(* IEC 61131-3 sources: std_i2980_v2.06_cp053/Source/IMM/ieccontrol/system (part 3) *)

(* ---- ABRuntimeMonitoring.pu ---- *)
(*
@h    ! WARNING !
@h    The Kemro K2 system (including software) only meets category B according to EN 954-1,
@h    thus it is not intended for usage in safety-relevant control applications in the field
@h    of personal safety (e.g. emergency stop).
@h    To implement potentially necessary safety-relevant control tasks, always use additional
@h    external safety devices that are intended for the particular purpose, and meet the necessary
@h    functional safety.
@h    For further information see EN 954-1 (EN ISO 13849-1) and/or the K2-x00 user manual, chapter
@h    "CE conformity, directives and standards".

This AB reacts on changes of sv_DataState and ODC1.sv_iInitOk
If sv_DataState is not nReady (this means reading or writing of data is in progress),
the runtime monitoring of the IEC - tasks will be switched off.
After sv_DataState changes to nReady again, the runtime monitoring will be switched on.
If the IEC - project is executed on Windows the runtime monitoring is switched off all the time.
The creation of the machine sequence, calculation of safety conditions, .... runs in TaskMid
To avoid cycle overflows during this procedure, the supervision is set to a higher value
during sequence creation.
Attention:
The supervision of TaskMid during creation of sequence should not be disabled so that
endless loops can be detected.
*)

IMPORT_OVER_LISTFILE
 SET_MAXIMUM_ACTIVE_INTERVAL
, tnDataState
, KCAT_HandleData
, KCAT_Status
, KSYS_Status

END_IMPORT

ALGORITHM_BLOCK ABRuntimeMonitoring #DUMMY_EDIT_BLOCK

SYSTEM_VAR
 sv_DataState : tnDataState (* indicates the state of xml handling (set by hmi) *);
 sv_bInitDone : BOOL;
 sv_bAllPUTasksExecuted : BOOL;
 sv_bInitStart : BOOL;
 sv_iActiveParamTransfers : DINT (* number of actually active parameter transfers (written by ABDriveParam.pu) *);
 sv_iReadMachineDataCount : UDINT (* counter which is increased after every loading of machine data  *);
 sv_iReadMoldDataCount : UDINT (* counter which is increased after every loading of mold data  *);
END_VAR

SYSTEM_OBJECT
 TaskException : TASK;
 TaskInject : TASK;
 TaskAnalog : TASK;
 TaskMid : TASK;
 TaskSequencer : TASK;
 PU_Task_13 : TASK;
 PU_Task_7 : TASK;
 PU_Task_3 : TASK;
 EV_Task_3 : TASK;
 EV_Task_7 : TASK;
 TaskHeating : TASK;
END_OBJECT

VAR
 mpiSequenceCreateState : REFTO DINT (* 0 nothing initialized, 10 sequence array initialized, 20 sequence array + safety initialized *);
 mbTaskPU13 : BOOL := FALSE;
 mbTaskPU7 : BOOL := FALSE;
 mbTaskPU3 : BOOL := FALSE;
 mbTaskEV3 : BOOL := FALSE;
 mbTaskEV7 : BOOL := FALSE;
END_VAR

POSTUPDATE_ALGORITHM pActivateDeactivate ON TaskException WITH sv_DataState,sv_bInitDone,mpiSequenceCreateState^,sv_iActiveParamTransfers

VAR
 StatusName : KCAT_HandleData;
 Name : STRING(255);
 Status : KCAT_Status;
 sValue : STRING(255);
 bIsWinNT : BOOL;
 bInitDone : BOOL;
 state : KSYS_Status;
 dSetInterval : TIME;
 bODC : BOOL;
 dSetTrigger : DINT;
END_VAR
#BEGIN_EDIT_BLOCK
(**************************************** WARNING ********************************************
 *** The KEBA Kemro K2 System including software is not intended for safety control tasks! ***
 ***                       For further information see Comment tab!                        ***
 *********************************************************************************************)

IF NOT bInitDone THEN
   Name := 'UOS.System';
   StatusName := KCAT_GetHandle(Name);
   IF StatusName.Status = KCAT_Status_OK THEN
      Status := KCAT_GetValue(Handle := StatusName.Handle, Buffer := sValue);
      IF (sValue = 'WINNT') THEN
         bIsWinNT := TRUE;
      ELSE
         bIsWinNT := FALSE;
      END_IF;
   END_IF;

   //get reference to state variable of sequence creation
   mpiSequenceCreateState := GET_SYNC_REFTO('ODC1.sv_iInitOK', T#0s, state);
   bODC := (state = KSYS_Status_OK);

   bInitDone := TRUE;
END_IF;

IF bIsWinNT THEN
   //don´t activate runtime monitoring if application is running on a pc
   RETURN;
END_IF;

IF bODC AND (mpiSequenceCreateState^ <> 20) THEN
   //creating of sequence in progress
   //creation of sequence, calculation of safety conditions, .... runs in TaskMid
   //-> set supervision to a higher value to avoid cycle overflows
   //supervision of TaskMid should not be disabled to detect endless loops
   dSetInterval := SET_MAXIMUM_ACTIVE_INTERVAL(TaskInject, GET_TASK_INTERVAL(TaskInject) * 10);
   dSetInterval := SET_MAXIMUM_ACTIVE_INTERVAL(TaskAnalog, GET_TASK_INTERVAL(TaskAnalog) * 10);
   dSetInterval := SET_MAXIMUM_ACTIVE_INTERVAL(TaskSequencer, GET_TASK_INTERVAL(TaskSequencer) * 10);
   dSetInterval := SET_MAXIMUM_ACTIVE_INTERVAL(TaskMid, GET_TASK_INTERVAL(TaskMid) * 200);

ELSIF sv_DataState <> nReady THEN
   //deactivate task runtime monitoring
   //if reading or writing of data is in progress
   dSetInterval := SET_MAXIMUM_ACTIVE_INTERVAL(TaskInject, T#0ms);
   dSetInterval := SET_MAXIMUM_ACTIVE_INTERVAL(TaskAnalog, T#0ms);
   dSetInterval := SET_MAXIMUM_ACTIVE_INTERVAL(TaskSequencer, T#0ms);
   dSetInterval := SET_MAXIMUM_ACTIVE_INTERVAL(TaskMid, T#0ms);

ELSIF sv_iActiveParamTransfers > 0 THEN
   //at least one paramter transfer is in progress -> increase maximum active interval of TaskMid
   dSetInterval := SET_MAXIMUM_ACTIVE_INTERVAL(TaskInject, GET_TASK_INTERVAL(TaskInject) * 10);
   dSetInterval := SET_MAXIMUM_ACTIVE_INTERVAL(TaskAnalog, GET_TASK_INTERVAL(TaskAnalog) * 10);
   dSetInterval := SET_MAXIMUM_ACTIVE_INTERVAL(TaskSequencer, GET_TASK_INTERVAL(TaskSequencer) * 10);
   dSetInterval := SET_MAXIMUM_ACTIVE_INTERVAL(TaskMid, GET_TASK_INTERVAL(TaskMid) * 200);

ELSE
   //activate task runtime monitoring
   dSetInterval := SET_MAXIMUM_ACTIVE_INTERVAL(TaskInject, GET_TASK_INTERVAL(TaskInject) * 10);
   dSetInterval := SET_MAXIMUM_ACTIVE_INTERVAL(TaskAnalog, GET_TASK_INTERVAL(TaskAnalog) * 10);
   dSetInterval := SET_MAXIMUM_ACTIVE_INTERVAL(TaskSequencer, GET_TASK_INTERVAL(TaskSequencer) * 10);
   dSetInterval := SET_MAXIMUM_ACTIVE_INTERVAL(TaskMid, GET_TASK_INTERVAL(TaskMid) * 10);
   dSetInterval := SET_MAXIMUM_ACTIVE_INTERVAL(TaskHeating, GET_TASK_INTERVAL(TaskHeating) * 10);

   dSetTrigger := SET_MAXIMUM_ACTIVE_TRIGGER(TaskHeating, 10);
END_IF;

;#END_EDIT_BLOCK END_ALGORITHM

(*
@h    ! WARNING !
@h    The Kemro K2 system (including software) only meets category B according to EN 954-1,
@h    thus it is not intended for usage in safety-relevant control applications in the field
@h    of personal safety (e.g. emergency stop).
@h    To implement potentially necessary safety-relevant control tasks, always use additional
@h    external safety devices that are intended for the particular purpose, and meet the necessary
@h    functional safety.
@h    For further information see EN 954-1 (EN ISO 13849-1) and/or the K2-x00 user manual, chapter
@h    "CE conformity, directives and standards".
*)

POSTUPDATE_ALGORITHM pTaskPU13 ON PU_Task_13(2147483653) WITH sv_bInitStart

#BEGIN_EDIT_BLOCK
(**************************************** WARNING ********************************************
 *** The KEBA Kemro K2 System including software is not intended for safety control tasks! ***
 ***                       For further information see Comment tab!                        ***
 *********************************************************************************************)

mbTaskPU13 := TRUE;

;#END_EDIT_BLOCK END_ALGORITHM

(*
@h    ! WARNING !
@h    The Kemro K2 system (including software) only meets category B according to EN 954-1,
@h    thus it is not intended for usage in safety-relevant control applications in the field
@h    of personal safety (e.g. emergency stop).
@h    To implement potentially necessary safety-relevant control tasks, always use additional
@h    external safety devices that are intended for the particular purpose, and meet the necessary
@h    functional safety.
@h    For further information see EN 954-1 (EN ISO 13849-1) and/or the K2-x00 user manual, chapter
@h    "CE conformity, directives and standards".
*)

POSTUPDATE_ALGORITHM pTaskPU7 ON PU_Task_7(2147483653) WITH sv_bInitStart

#BEGIN_EDIT_BLOCK
(**************************************** WARNING ********************************************
 *** The KEBA Kemro K2 System including software is not intended for safety control tasks! ***
 ***                       For further information see Comment tab!                        ***
 *********************************************************************************************)

mbTaskPU7 := TRUE;

;#END_EDIT_BLOCK END_ALGORITHM

(*
@h    ! WARNING !
@h    The Kemro K2 system (including software) only meets category B according to EN 954-1,
@h    thus it is not intended for usage in safety-relevant control applications in the field
@h    of personal safety (e.g. emergency stop).
@h    To implement potentially necessary safety-relevant control tasks, always use additional
@h    external safety devices that are intended for the particular purpose, and meet the necessary
@h    functional safety.
@h    For further information see EN 954-1 (EN ISO 13849-1) and/or the K2-x00 user manual, chapter
@h    "CE conformity, directives and standards".
*)

POSTUPDATE_ALGORITHM pTaskPU3 ON PU_Task_3(2147483653) WITH sv_bInitStart

#BEGIN_EDIT_BLOCK
(**************************************** WARNING ********************************************
 *** The KEBA Kemro K2 System including software is not intended for safety control tasks! ***
 ***                       For further information see Comment tab!                        ***
 *********************************************************************************************)

mbTaskPU3 := TRUE;

;#END_EDIT_BLOCK END_ALGORITHM

(*
@h    ! WARNING !
@h    The Kemro K2 system (including software) only meets category B according to EN 954-1,
@h    thus it is not intended for usage in safety-relevant control applications in the field
@h    of personal safety (e.g. emergency stop).
@h    To implement potentially necessary safety-relevant control tasks, always use additional
@h    external safety devices that are intended for the particular purpose, and meet the necessary
@h    functional safety.
@h    For further information see EN 954-1 (EN ISO 13849-1) and/or the K2-x00 user manual, chapter
@h    "CE conformity, directives and standards".
*)

POSTUPDATE_ALGORITHM pTaskEV3 ON EV_Task_3(2147483653) WITH sv_bInitStart

#BEGIN_EDIT_BLOCK
(**************************************** WARNING ********************************************
 *** The KEBA Kemro K2 System including software is not intended for safety control tasks! ***
 ***                       For further information see Comment tab!                        ***
 *********************************************************************************************)

mbTaskEV3 := TRUE;

;#END_EDIT_BLOCK END_ALGORITHM

(*
@h    ! WARNING !
@h    The Kemro K2 system (including software) only meets category B according to EN 954-1,
@h    thus it is not intended for usage in safety-relevant control applications in the field
@h    of personal safety (e.g. emergency stop).
@h    To implement potentially necessary safety-relevant control tasks, always use additional
@h    external safety devices that are intended for the particular purpose, and meet the necessary
@h    functional safety.
@h    For further information see EN 954-1 (EN ISO 13849-1) and/or the K2-x00 user manual, chapter
@h    "CE conformity, directives and standards".
*)

POSTUPDATE_ALGORITHM pTaskEV7 ON EV_Task_7(2147483653) WITH sv_bInitStart

#BEGIN_EDIT_BLOCK
(**************************************** WARNING ********************************************
 *** The KEBA Kemro K2 System including software is not intended for safety control tasks! ***
 ***                       For further information see Comment tab!                        ***
 *********************************************************************************************)

mbTaskEV7 := TRUE;

;#END_EDIT_BLOCK END_ALGORITHM

PROCESS_ALGORITHM paCheckExecutedTasks ON TaskMid AUTOSTART

#BEGIN_EDIT_BLOCK
(**************************************** WARNING ********************************************
 *** The KEBA Kemro K2 System including software is not intended for safety control tasks! ***
 ***                       For further information see Comment tab!                        ***
 *********************************************************************************************)

IF mbTaskEV3 AND mbTaskEV7 AND mbTaskPU13 AND mbTaskPU3 AND mbTaskPU7 THEN
   //set SV for ABMovementRegister to signalize that sv_bInitStart is TRUE
   //and all relevant postupdate tasks and event tasks are executed at least one time
   sv_bAllPUTasksExecuted := TRUE;
   STOP_PROCESS_ALGORITHM();
END_IF;

;#END_EDIT_BLOCK END_ALGORITHM

POSTUPDATE_ALGORITHM pDataState ON PU_Task_3(1) WITH sv_DataState

VAR
 oldDataState : tnDataState;
END_VAR
#BEGIN_EDIT_BLOCK
(**************************************** WARNING ********************************************
 *** The KEBA Kemro K2 System including software is not intended for safety control tasks! ***
 ***                       For further information see Comment tab!                        ***
 *********************************************************************************************)

IF (sv_DataState = nReady) THEN
   IF (oldDataState = nReadMachineData) THEN
      sv_iReadMachineDataCount := sv_iReadMachineDataCount + 1;
   ELSIF oldDataState = nReadMoldData THEN
      sv_iReadMoldDataCount := sv_iReadMoldDataCount + 1;
   END_IF;
END_IF;

oldDataState := sv_DataState;

;#END_EDIT_BLOCK END_ALGORITHM

END_ALGORITHM_BLOCK

#END_OF_IEC_PART

@Puma @IecEditor 6 68 @Pou 25
@@@BEG_Comment@@@
@h    ! WARNING !
@h    The Kemro K2 system (including software) only meets category B according to EN 954-1,
@h    thus it is not intended for usage in safety-relevant control applications in the field
@h    of personal safety (e.g. emergency stop).
@h    To implement potentially necessary safety-relevant control tasks, always use additional
@h    external safety devices that are intended for the particular purpose, and meet the necessary
@h    functional safety.
@h    For further information see EN 954-1 (EN ISO 13849-1) and/or the K2-x00 user manual, chapter
@h    "CE conformity, directives and standards".

This AB reacts on changes of sv_DataState and ODC1.sv_iInitOk
If sv_DataState is not nReady (this means reading or writing of data is in progress),
the runtime monitoring of the IEC - tasks will be switched off.
After sv_DataState changes to nReady again, the runtime monitoring will be switched on.
If the IEC - project is executed on Windows the runtime monitoring is switched off all the time.
The creation of the machine sequence, calculation of safety conditions, .... runs in TaskMid
To avoid cycle overflows during this procedure, the supervision is set to a higher value
during sequence creation.
Attention:
The supervision of TaskMid during creation of sequence should not be disabled so that
endless loops can be detected.
@@@END_Comment@@@

@BEG_Contents

@BEG_Func
@RT(17)FuncTreeContainer
1
@Var @RT(27)SET_MAXIMUM_ACTIVE_INTERVAL @RT(0) @T @T @DERIVED 0 @F @RT(22)KEBA_STANDARD_FUNCTION @F
@T
@BEG_Attrib
0 @RT(0) @RT(0)
@END_Attrib
1 1 @F @F @F @F

@END_Func

@BEG_Const
@RT(18)ConstTreeContainer
0
@END_Const

@BEG_Export

@BEG_Kind
@ALGORITHM_BLOCK @RT(19)ABRuntimeMonitoring @STRUCTURED_TEXT
@RT(0) @RT(0) @RT(0)
@END_Kind

@BEG_Dcl
@RT(16)DclTreeContainer
24
@Var @RT(13)TaskException @RT(0) @T @F @DT @RT(4)TASK @RT(0) @T @T @BASIC 0 @F
@F @F
@T
@BEG_Attrib
3 @RT(0) @RT(0) @RT(0)
@END_Attrib
1 7 @F @F @F @F

@Var @RT(12)sv_DataState @RT(0) @T @T @DERIVED 0 @T @T @DT @RT(11)tnDataState @RT(0) @T @T @UNKNOWN 0 @F
@F @F
@T
@BEG_Attrib
3 @RT(0) @RT(48)indicates the state of xml handling (set by hmi) @RT(0)
@END_Attrib
1 8 @F @F @F @F

@Var @RT(12)sv_bInitDone @RT(0) @T @F @DT @RT(4)BOOL @RT(0) @T @T @BASIC 0 @F
@F @F
@T
@BEG_Attrib
3 @RT(0) @RT(0) @RT(0)
@END_Attrib
1 8 @F @F @F @F

@Var @RT(22)mpiSequenceCreateState @RT(0) @T @T @REFTO 0 @T @DT @RT(4)DINT @RT(0) @T @T @BASIC 0 @F
@F @F
@T
@BEG_Attrib
3 @RT(0) @RT(92)0 nothing initialized, 10 sequence array initialized, 20 sequence array + safety initialized @RT(0)
@END_Attrib
1 0 @F @F @F @F

@Var @RT(10)TaskInject @RT(0) @T @F @DT @RT(4)TASK @RT(0) @T @T @BASIC 0 @F
@F @F
@T
@BEG_Attrib
3 @RT(0) @RT(0) @RT(0)
@END_Attrib
1 7 @F @F @F @F

@Var @RT(10)TaskAnalog @RT(0) @T @F @DT @RT(4)TASK @RT(0) @T @T @BASIC 0 @F
@F @F
@T
@BEG_Attrib
3 @RT(0) @RT(0) @RT(0)
@END_Attrib
1 7 @F @F @F @F

@Var @RT(7)TaskMid @RT(0) @T @F @DT @RT(4)TASK @RT(0) @T @T @BASIC 0 @F
@F @F
@T
@BEG_Attrib
3 @RT(0) @RT(0) @RT(0)
@END_Attrib
1 7 @F @F @F @F

@Var @RT(13)TaskSequencer @RT(0) @T @F @DT @RT(4)TASK @RT(0) @T @T @BASIC 0 @F
@F @F
@T
@BEG_Attrib
3 @RT(0) @RT(0) @RT(0)
@END_Attrib
1 7 @F @F @F @F

@Var @RT(10)mbTaskPU13 @RT(0) @T @F @DT @RT(4)BOOL @RT(0) @T @T @BASIC 0 @F
@F @F
@T
@BEG_Attrib
3 @RT(5)FALSE @RT(0) @RT(0)
@END_Attrib
1 0 @F @F @F @F

@Var @RT(9)mbTaskPU7 @RT(0) @T @F @DT @RT(4)BOOL @RT(0) @T @T @BASIC 0 @F
@F @F
@T
@BEG_Attrib
3 @RT(5)FALSE @RT(0) @RT(0)
@END_Attrib
1 0 @F @F @F @F

@Var @RT(9)mbTaskPU3 @RT(0) @T @F @DT @RT(4)BOOL @RT(0) @T @T @BASIC 0 @F
@F @F
@T
@BEG_Attrib
3 @RT(5)FALSE @RT(0) @RT(0)
@END_Attrib
1 0 @F @F @F @F

@Var @RT(9)mbTaskEV3 @RT(0) @T @F @DT @RT(4)BOOL @RT(0) @T @T @BASIC 0 @F
@F @F
@T
@BEG_Attrib
3 @RT(5)FALSE @RT(0) @RT(0)
@END_Attrib
1 0 @F @F @F @F

@Var @RT(9)mbTaskEV7 @RT(0) @T @F @DT @RT(4)BOOL @RT(0) @T @T @BASIC 0 @F
@F @F
@T
@BEG_Attrib
3 @RT(5)FALSE @RT(0) @RT(0)
@END_Attrib
1 0 @F @F @F @F

@Var @RT(22)sv_bAllPUTasksExecuted @RT(0) @T @F @DT @RT(4)BOOL @RT(0) @T @T @BASIC 0 @F
@F @F
@T
@BEG_Attrib
3 @RT(0) @RT(0) @RT(0)
@END_Attrib
1 8 @F @F @F @F

@Var @RT(13)sv_bInitStart @RT(0) @T @F @DT @RT(4)BOOL @RT(0) @T @T @BASIC 0 @F
@F @F
@T
@BEG_Attrib
3 @RT(0) @RT(0) @RT(0)
@END_Attrib
1 8 @F @F @F @F

@Var @RT(10)PU_Task_13 @RT(0) @T @F @DT @RT(4)TASK @RT(0) @T @T @BASIC 0 @F
@F @F
@T
@BEG_Attrib
3 @RT(0) @RT(0) @RT(0)
@END_Attrib
1 7 @F @F @F @F

@Var @RT(9)PU_Task_7 @RT(0) @T @F @DT @RT(4)TASK @RT(0) @T @T @BASIC 0 @F
@F @F
@T
@BEG_Attrib
3 @RT(0) @RT(0) @RT(0)
@END_Attrib
1 7 @F @F @F @F

@Var @RT(9)PU_Task_3 @RT(0) @T @F @DT @RT(4)TASK @RT(0) @T @T @BASIC 0 @F
@F @F
@T
@BEG_Attrib
3 @RT(0) @RT(0) @RT(0)
@END_Attrib
1 7 @F @F @F @F

@Var @RT(9)EV_Task_3 @RT(0) @T @F @DT @RT(4)TASK @RT(0) @T @T @BASIC 0 @F
@F @F
@T
@BEG_Attrib
3 @RT(0) @RT(0) @RT(0)
@END_Attrib
1 7 @F @F @F @F

@Var @RT(9)EV_Task_7 @RT(0) @T @F @DT @RT(4)TASK @RT(0) @T @T @BASIC 0 @F
@F @F
@T
@BEG_Attrib
3 @RT(0) @RT(0) @RT(0)
@END_Attrib
1 7 @F @F @F @F

@Var @RT(24)sv_iActiveParamTransfers @RT(0) @T @F @DT @RT(4)DINT @RT(0) @T @T @BASIC 0 @F
@F @F
@T
@BEG_Attrib
3 @RT(0) @RT(74)number of actually active parameter transfers (written by ABDriveParam.pu) @RT(0)
@END_Attrib
1 8 @F @F @F @F

@Var @RT(11)TaskHeating @RT(0) @T @F @DT @RT(4)TASK @RT(0) @T @T @BASIC 0 @F
@F @F
@T
@BEG_Attrib
3 @RT(0) @RT(0) @RT(0)
@END_Attrib
1 7 @F @F @F @F

@Var @RT(24)sv_iReadMachineDataCount @RT(0) @T @F @DT @RT(5)UDINT @RT(0) @T @T @BASIC 0 @F
@F @F
@T
@BEG_Attrib
3 @RT(0) @RT(63)counter which is increased after every loading of machine data  @RT(0)
@END_Attrib
1 8 @F @F @F @F

@Var @RT(21)sv_iReadMoldDataCount @RT(0) @T @F @DT @RT(5)UDINT @RT(0) @T @T @BASIC 0 @F
@F @F
@T
@BEG_Attrib
3 @RT(0) @RT(60)counter which is increased after every loading of mold data  @RT(0)
@END_Attrib
1 8 @F @F @F @F

@END_Dcl

@END_Export

@BEG_Body

8

@BEG_Export

@BEG_Algo
@POSTUPDATE_ALGORITHM @RT(19)pActivateDeactivate @STRUCTURED_TEXT
@RT(0) @RT(74)sv_DataState,sv_bInitDone,mpiSequenceCreateState^,sv_iActiveParamTransfers @RT(13)TaskException @F @F
@END_Algo

@BEG_Dcl
@RT(16)DclTreeContainer
10
@Var @RT(10)StatusName @RT(0) @T @T @DERIVED 0 @T @T @DT @RT(15)KCAT_HandleData @RT(0) @T @T @UNKNOWN 0 @F
@F @F
@T
@BEG_Attrib
3 @RT(0) @RT(0) @RT(0)
@END_Attrib
1 0 @F @F @F @F

@Var @RT(4)Name @RT(0) @T @F @DT @RT(11)STRING(255) @RT(0) @T @T @STRING 0 @F @RT(3)255 @F
@F @F
@T
@BEG_Attrib
3 @RT(0) @RT(0) @RT(0)
@END_Attrib
1 0 @F @F @F @F

@Var @RT(6)Status @RT(0) @T @T @DERIVED 0 @T @T @DT @RT(11)KCAT_Status @RT(0) @T @T @UNKNOWN 0 @F
@F @F
@T
@BEG_Attrib
3 @RT(0) @RT(0) @RT(0)
@END_Attrib
1 0 @F @F @F @F

@Var @RT(6)sValue @RT(0) @T @F @DT @RT(11)STRING(255) @RT(0) @T @T @STRING 0 @F @RT(3)255 @F
@F @F
@T
@BEG_Attrib
3 @RT(0) @RT(0) @RT(0)
@END_Attrib
1 0 @F @F @F @F

@Var @RT(8)bIsWinNT @RT(0) @T @F @DT @RT(4)BOOL @RT(0) @T @T @BASIC 0 @F
@F @F
@T
@BEG_Attrib
3 @RT(0) @RT(0) @RT(0)
@END_Attrib
1 0 @F @F @F @F

@Var @RT(9)bInitDone @RT(0) @T @F @DT @RT(4)BOOL @RT(0) @T @T @BASIC 0 @F
@F @F
@T
@BEG_Attrib
3 @RT(0) @RT(0) @RT(0)
@END_Attrib
1 0 @F @F @F @F

@Var @RT(5)state @RT(0) @T @T @DERIVED 0 @T @T @DT @RT(11)KSYS_Status @RT(0) @T @T @UNKNOWN 0 @F
@F @F
@T
@BEG_Attrib
3 @RT(0) @RT(0) @RT(0)
@END_Attrib
1 0 @F @F @F @F

@Var @RT(12)dSetInterval @RT(0) @T @F @DT @RT(4)TIME @RT(0) @T @T @BASIC 0 @F
@F @F
@T
@BEG_Attrib
3 @RT(0) @RT(0) @RT(0)
@END_Attrib
1 0 @F @F @F @F

@Var @RT(4)bODC @RT(0) @T @F @DT @RT(4)BOOL @RT(0) @T @T @BASIC 0 @F
@F @F
@T
@BEG_Attrib
3 @RT(0) @RT(0) @RT(0)
@END_Attrib
1 0 @F @F @F @F

@Var @RT(11)dSetTrigger @RT(0) @T @F @DT @RT(4)DINT @RT(0) @T @T @BASIC 0 @F
@F @F
@T
@BEG_Attrib
3 @RT(0) @RT(0) @RT(0)
@END_Attrib
1 0 @F @F @F @F

@END_Dcl

@END_Export

@BEG_Export

@BEG_Algo
@POSTUPDATE_ALGORITHM @RT(9)pTaskPU13 @STRUCTURED_TEXT
@RT(0) @RT(13)sv_bInitStart @RT(22)PU_Task_13(2147483653) @F @F
@END_Algo

@BEG_Dcl
@RT(16)DclTreeContainer
0
@END_Dcl

@END_Export

@BEG_Export

@BEG_Algo
@POSTUPDATE_ALGORITHM @RT(8)pTaskPU7 @STRUCTURED_TEXT
@RT(0) @RT(13)sv_bInitStart @RT(21)PU_Task_7(2147483653) @F @F
@END_Algo

@BEG_Dcl
@RT(16)DclTreeContainer
0
@END_Dcl

@END_Export

@BEG_Export

@BEG_Algo
@POSTUPDATE_ALGORITHM @RT(8)pTaskPU3 @STRUCTURED_TEXT
@RT(0) @RT(13)sv_bInitStart @RT(21)PU_Task_3(2147483653) @F @F
@END_Algo

@BEG_Dcl
@RT(16)DclTreeContainer
0
@END_Dcl

@END_Export

@BEG_Export

@BEG_Algo
@POSTUPDATE_ALGORITHM @RT(8)pTaskEV3 @STRUCTURED_TEXT
@RT(0) @RT(13)sv_bInitStart @RT(21)EV_Task_3(2147483653) @F @F
@END_Algo

@BEG_Dcl
@RT(16)DclTreeContainer
0
@END_Dcl

@END_Export

@BEG_Export

@BEG_Algo
@POSTUPDATE_ALGORITHM @RT(8)pTaskEV7 @STRUCTURED_TEXT
@RT(0) @RT(13)sv_bInitStart @RT(21)EV_Task_7(2147483653) @F @F
@END_Algo

@BEG_Dcl
@RT(16)DclTreeContainer
0
@END_Dcl

@END_Export

@BEG_Export

@BEG_Algo
@PROCESS_ALGORITHM @RT(20)paCheckExecutedTasks @STRUCTURED_TEXT
@RT(0) @RT(0) @RT(7)TaskMid @T @F
@END_Algo

@BEG_Dcl
@RT(16)DclTreeContainer
0
@END_Dcl

@END_Export

@BEG_Export

@BEG_Algo
@POSTUPDATE_ALGORITHM @RT(10)pDataState @STRUCTURED_TEXT
@RT(0) @RT(12)sv_DataState @RT(12)PU_Task_3(1) @F @F
@END_Algo

@BEG_Dcl
@RT(16)DclTreeContainer
1
@Var @RT(12)oldDataState @RT(0) @T @T @DERIVED 0 @F @RT(11)tnDataState @F
@T
@BEG_Attrib
3 @RT(0) @RT(0) @RT(0)
@END_Attrib
1 0 @F @F @F @F

@END_Dcl

@END_Export

@BEG_Body
@TL(67)
(**************************************** WARNING ********************************************
 *** The KEBA Kemro K2 System including software is not intended for safety control tasks! ***
 ***                       For further information see Comment tab!                        ***
 *********************************************************************************************)

IF NOT bInitDone THEN
   Name := 'UOS.System';
   StatusName := KCAT_GetHandle(Name);
   IF StatusName.Status = KCAT_Status_OK THEN
      Status := KCAT_GetValue(Handle := StatusName.Handle, Buffer := sValue);
      IF (sValue = 'WINNT') THEN
         bIsWinNT := TRUE;
      ELSE
         bIsWinNT := FALSE;
      END_IF;
   END_IF;

   //get reference to state variable of sequence creation
   mpiSequenceCreateState := GET_SYNC_REFTO('ODC1.sv_iInitOK', T#0s, state);
   bODC := (state = KSYS_Status_OK);

   bInitDone := TRUE;
END_IF;

IF bIsWinNT THEN
   //don´t activate runtime monitoring if application is running on a pc
   RETURN;
END_IF;

IF bODC AND (mpiSequenceCreateState^ <> 20) THEN
   //creating of sequence in progress
   //creation of sequence, calculation of safety conditions, .... runs in TaskMid
   //-> set supervision to a higher value to avoid cycle overflows
   //supervision of TaskMid should not be disabled to detect endless loops
   dSetInterval := SET_MAXIMUM_ACTIVE_INTERVAL(TaskInject, GET_TASK_INTERVAL(TaskInject) * 10);
   dSetInterval := SET_MAXIMUM_ACTIVE_INTERVAL(TaskAnalog, GET_TASK_INTERVAL(TaskAnalog) * 10);
   dSetInterval := SET_MAXIMUM_ACTIVE_INTERVAL(TaskSequencer, GET_TASK_INTERVAL(TaskSequencer) * 10);
   dSetInterval := SET_MAXIMUM_ACTIVE_INTERVAL(TaskMid, GET_TASK_INTERVAL(TaskMid) * 200);

ELSIF sv_DataState <> nReady THEN
   //deactivate task runtime monitoring
   //if reading or writing of data is in progress
   dSetInterval := SET_MAXIMUM_ACTIVE_INTERVAL(TaskInject, T#0ms);
   dSetInterval := SET_MAXIMUM_ACTIVE_INTERVAL(TaskAnalog, T#0ms);
   dSetInterval := SET_MAXIMUM_ACTIVE_INTERVAL(TaskSequencer, T#0ms);
   dSetInterval := SET_MAXIMUM_ACTIVE_INTERVAL(TaskMid, T#0ms);

ELSIF sv_iActiveParamTransfers > 0 THEN
   //at least one paramter transfer is in progress -> increase maximum active interval of TaskMid
   dSetInterval := SET_MAXIMUM_ACTIVE_INTERVAL(TaskInject, GET_TASK_INTERVAL(TaskInject) * 10);
   dSetInterval := SET_MAXIMUM_ACTIVE_INTERVAL(TaskAnalog, GET_TASK_INTERVAL(TaskAnalog) * 10);
   dSetInterval := SET_MAXIMUM_ACTIVE_INTERVAL(TaskSequencer, GET_TASK_INTERVAL(TaskSequencer) * 10);
   dSetInterval := SET_MAXIMUM_ACTIVE_INTERVAL(TaskMid, GET_TASK_INTERVAL(TaskMid) * 200);

ELSE
   //activate task runtime monitoring
   dSetInterval := SET_MAXIMUM_ACTIVE_INTERVAL(TaskInject, GET_TASK_INTERVAL(TaskInject) * 10);
   dSetInterval := SET_MAXIMUM_ACTIVE_INTERVAL(TaskAnalog, GET_TASK_INTERVAL(TaskAnalog) * 10);
   dSetInterval := SET_MAXIMUM_ACTIVE_INTERVAL(TaskSequencer, GET_TASK_INTERVAL(TaskSequencer) * 10);
   dSetInterval := SET_MAXIMUM_ACTIVE_INTERVAL(TaskMid, GET_TASK_INTERVAL(TaskMid) * 10);
   dSetInterval := SET_MAXIMUM_ACTIVE_INTERVAL(TaskHeating, GET_TASK_INTERVAL(TaskHeating) * 10);

   dSetTrigger := SET_MAXIMUM_ACTIVE_TRIGGER(TaskHeating, 10);
END_IF;

@END_Body

@@@BEG_Comment@@@
@TL(0)

@@@END_Comment@@@

@BEG_Body
@TL(7)
(**************************************** WARNING ********************************************
 *** The KEBA Kemro K2 System including software is not intended for safety control tasks! ***
 ***                       For further information see Comment tab!                        ***
 *********************************************************************************************)

mbTaskPU13 := TRUE;

@END_Body

@@@BEG_Comment@@@
@TL(9)
@h    ! WARNING !
@h    The Kemro K2 system (including software) only meets category B according to EN 954-1,
@h    thus it is not intended for usage in safety-relevant control applications in the field
@h    of personal safety (e.g. emergency stop).
@h    To implement potentially necessary safety-relevant control tasks, always use additional
@h    external safety devices that are intended for the particular purpose, and meet the necessary
@h    functional safety.
@h    For further information see EN 954-1 (EN ISO 13849-1) and/or the K2-x00 user manual, chapter
@h    "CE conformity, directives and standards".
@@@END_Comment@@@

@BEG_Body
@TL(7)
(**************************************** WARNING ********************************************
 *** The KEBA Kemro K2 System including software is not intended for safety control tasks! ***
 ***                       For further information see Comment tab!                        ***
 *********************************************************************************************)

mbTaskPU7 := TRUE;

@END_Body

@@@BEG_Comment@@@
@TL(9)
@h    ! WARNING !
@h    The Kemro K2 system (including software) only meets category B according to EN 954-1,
@h    thus it is not intended for usage in safety-relevant control applications in the field
@h    of personal safety (e.g. emergency stop).
@h    To implement potentially necessary safety-relevant control tasks, always use additional
@h    external safety devices that are intended for the particular purpose, and meet the necessary
@h    functional safety.
@h    For further information see EN 954-1 (EN ISO 13849-1) and/or the K2-x00 user manual, chapter
@h    "CE conformity, directives and standards".
@@@END_Comment@@@

@BEG_Body
@TL(7)
(**************************************** WARNING ********************************************
 *** The KEBA Kemro K2 System including software is not intended for safety control tasks! ***
 ***                       For further information see Comment tab!                        ***
 *********************************************************************************************)

mbTaskPU3 := TRUE;

@END_Body

@@@BEG_Comment@@@
@TL(9)
@h    ! WARNING !
@h    The Kemro K2 system (including software) only meets category B according to EN 954-1,
@h    thus it is not intended for usage in safety-relevant control applications in the field
@h    of personal safety (e.g. emergency stop).
@h    To implement potentially necessary safety-relevant control tasks, always use additional
@h    external safety devices that are intended for the particular purpose, and meet the necessary
@h    functional safety.
@h    For further information see EN 954-1 (EN ISO 13849-1) and/or the K2-x00 user manual, chapter
@h    "CE conformity, directives and standards".
@@@END_Comment@@@

@BEG_Body
@TL(7)
(**************************************** WARNING ********************************************
 *** The KEBA Kemro K2 System including software is not intended for safety control tasks! ***
 ***                       For further information see Comment tab!                        ***
 *********************************************************************************************)

mbTaskEV3 := TRUE;

@END_Body

@@@BEG_Comment@@@
@TL(9)
@h    ! WARNING !
@h    The Kemro K2 system (including software) only meets category B according to EN 954-1,
@h    thus it is not intended for usage in safety-relevant control applications in the field
@h    of personal safety (e.g. emergency stop).
@h    To implement potentially necessary safety-relevant control tasks, always use additional
@h    external safety devices that are intended for the particular purpose, and meet the necessary
@h    functional safety.
@h    For further information see EN 954-1 (EN ISO 13849-1) and/or the K2-x00 user manual, chapter
@h    "CE conformity, directives and standards".
@@@END_Comment@@@

@BEG_Body
@TL(7)
(**************************************** WARNING ********************************************
 *** The KEBA Kemro K2 System including software is not intended for safety control tasks! ***
 ***                       For further information see Comment tab!                        ***
 *********************************************************************************************)

mbTaskEV7 := TRUE;

@END_Body

@@@BEG_Comment@@@
@TL(9)
@h    ! WARNING !
@h    The Kemro K2 system (including software) only meets category B according to EN 954-1,
@h    thus it is not intended for usage in safety-relevant control applications in the field
@h    of personal safety (e.g. emergency stop).
@h    To implement potentially necessary safety-relevant control tasks, always use additional
@h    external safety devices that are intended for the particular purpose, and meet the necessary
@h    functional safety.
@h    For further information see EN 954-1 (EN ISO 13849-1) and/or the K2-x00 user manual, chapter
@h    "CE conformity, directives and standards".
@@@END_Comment@@@

@BEG_Body
@TL(12)
(**************************************** WARNING ********************************************
 *** The KEBA Kemro K2 System including software is not intended for safety control tasks! ***
 ***                       For further information see Comment tab!                        ***
 *********************************************************************************************)

IF mbTaskEV3 AND mbTaskEV7 AND mbTaskPU13 AND mbTaskPU3 AND mbTaskPU7 THEN
   //set SV for ABMovementRegister to signalize that sv_bInitStart is TRUE
   //and all relevant postupdate tasks and event tasks are executed at least one time
   sv_bAllPUTasksExecuted := TRUE;
   STOP_PROCESS_ALGORITHM();
END_IF;

@END_Body

@@@BEG_Comment@@@
@TL(0)

@@@END_Comment@@@

@BEG_Body
@TL(16)
(**************************************** WARNING ********************************************
 *** The KEBA Kemro K2 System including software is not intended for safety control tasks! ***
 ***                       For further information see Comment tab!                        ***
 *********************************************************************************************)

IF (sv_DataState = nReady) THEN
   IF (oldDataState = nReadMachineData) THEN
      sv_iReadMachineDataCount := sv_iReadMachineDataCount + 1;
   ELSIF oldDataState = nReadMoldData THEN
      sv_iReadMoldDataCount := sv_iReadMoldDataCount + 1;
   END_IF;
END_IF;

oldDataState := sv_DataState;

@END_Body

@@@BEG_Comment@@@
@TL(0)

@@@END_Comment@@@
@END_Body

@END_Contents

(* ---- ABUsbEvent.pu ---- *)
(*
@h    ! WARNING !
@h    The Kemro K2 system (including software) only meets category B according to EN 954-1,
@h    thus it is not intended for usage in safety-relevant control applications in the field
@h    of personal safety (e.g. emergency stop).
@h    To implement potentially necessary safety-relevant control tasks, always use additional
@h    external safety devices that are intended for the particular purpose, and meet the necessary
@h    functional safety.
@h    For further information see EN 954-1 (EN ISO 13849-1) and/or the K2-x00 user manual, chapter
@h    "CE conformity, directives and standards".

This algorithm block registers the systemevent system.evUsbEvent for callback on usb device attach/detach.

*)

IMPORT_OVER_LISTFILE
 IS_LINKED
, KPUSB_Event
, KPUSB_Notification

END_IMPORT

ALGORITHM_BLOCK ABUsbEvent #DUMMY_EDIT_BLOCK

SYSTEM_VAR
 sv_bInitDone : BOOL;
 sv_bMachineLockAvailable : BOOL;
END_VAR

SYSTEM_OBJECT
 TaskVis : TASK;
 evUsbEvent : KPUSB_Event;
END_OBJECT

VAR
 fbRegisterUsb : KPUSB_Notification;
END_VAR

POSTUPDATE_ALGORITHM pInit ON TaskVis WITH sv_bInitDone

#BEGIN_EDIT_BLOCK
(**************************************** WARNING ********************************************
 *** The KEBA Kemro K2 System including software is not intended for safety control tasks! ***
 ***                       For further information see Comment tab!                        ***
 *********************************************************************************************)

fbRegisterUsb(UseDeviceInfo := FALSE, Event := evUsbEvent);

;#END_EDIT_BLOCK END_ALGORITHM

END_ALGORITHM_BLOCK

#END_OF_IEC_PART

@Puma @IecEditor 6 131 @Pou 25
@@@BEG_Comment@@@
@h    ! WARNING !
@h    The Kemro K2 system (including software) only meets category B according to EN 954-1,
@h    thus it is not intended for usage in safety-relevant control applications in the field
@h    of personal safety (e.g. emergency stop).
@h    To implement potentially necessary safety-relevant control tasks, always use additional
@h    external safety devices that are intended for the particular purpose, and meet the necessary
@h    functional safety.
@h    For further information see EN 954-1 (EN ISO 13849-1) and/or the K2-x00 user manual, chapter
@h    "CE conformity, directives and standards".

This algorithm block registers the systemevent system.evUsbEvent for callback on usb device attach/detach.

@@@END_Comment@@@

@BEG_Contents

@BEG_Func
@RT(17)FuncTreeContainer
1
@Var @RT(9)IS_LINKED @RT(0) @T @T @DERIVED 0 @F @RT(22)KEBA_STANDARD_FUNCTION @F
@T
@BEG_Attrib
0 @RT(0) @RT(0)
@END_Attrib
1 1 @F @F @F @F

@END_Func

@BEG_Const
@RT(18)ConstTreeContainer
0
@END_Const

@BEG_Export

@BEG_Kind
@ALGORITHM_BLOCK @RT(10)ABUsbEvent @STRUCTURED_TEXT
@RT(0) @RT(0) @RT(0)
@END_Kind

@BEG_Dcl
@RT(16)DclTreeContainer
5
@Var @RT(7)TaskVis @RT(0) @T @T @RENAMED 0 @T @T @DT @RT(4)TASK @RT(0) @T @T @BASIC 0 @F
@F @F
@T
@BEG_Attrib
3 @RT(0) @RT(0) @RT(0)
@END_Attrib
1 7 @F @F @F @F

@Var @RT(10)evUsbEvent @RT(0) @T @T @DERIVED 0 @T @T @DT @RT(11)KPUSB_Event @RT(0) @T @T @UNKNOWN 0 @F
@F @F
@T
@BEG_Attrib
3 @RT(0) @RT(0) @RT(0)
@END_Attrib
1 7 @F @F @F @F

@Var @RT(12)sv_bInitDone @RT(0) @T @T @RENAMED 0 @T @T @DT @RT(4)BOOL @RT(0) @T @T @BASIC 0 @F
@F @F
@T
@BEG_Attrib
3 @RT(0) @RT(0) @RT(0)
@END_Attrib
1 8 @F @F @F @F

@Var @RT(24)sv_bMachineLockAvailable @RT(0) @T @F @DT @RT(4)BOOL @RT(0) @T @T @BASIC 0 @F
@F @F
@T
@BEG_Attrib
3 @RT(0) @RT(0) @RT(0)
@END_Attrib
1 8 @F @F @F @F

@Var @RT(13)fbRegisterUsb @RT(0) @T @T @DERIVED 0 @T @T @DT @RT(18)KPUSB_Notification @RT(0) @T @T @UNKNOWN 0 @F
@F @F
@T
@BEG_Attrib
3 @RT(0) @RT(0) @RT(0)
@END_Attrib
1 0 @F @F @F @F

@END_Dcl

@END_Export

@BEG_Body

1

@BEG_Export

@BEG_Algo
@POSTUPDATE_ALGORITHM @RT(5)pInit @STRUCTURED_TEXT
@RT(0) @RT(12)sv_bInitDone @RT(7)TaskVis @F @F
@END_Algo

@BEG_Dcl
@RT(16)DclTreeContainer
0
@END_Dcl

@END_Export

@BEG_Body
@TL(9)
(**************************************** WARNING ********************************************
 *** The KEBA Kemro K2 System including software is not intended for safety control tasks! ***
 ***                       For further information see Comment tab!                        ***
 *********************************************************************************************)

fbRegisterUsb(UseDeviceInfo := FALSE, Event := evUsbEvent);

@END_Body

@@@BEG_Comment@@@
@TL(0)

@@@END_Comment@@@
@END_Body

@END_Contents

(* ---- FPlausMaxInjectPressure.pu ---- *)
IMPORT_OVER_LISTFILE
 GET_SYNC_REFTO
, IS_LINKED
, tsLimitDataReal
, KSYS_Status
, KAPPL_LintabData
, tOptionId
, KAPPL_LintabData_2P

END_IMPORT

PLAUSIBILITY_FUNCTION FPlausMaxInjectPressure : tsLimitDataReal

VAR_INPUT
 DeviceClass : INT;
 Userlevel : INT;
END_VAR

VAR
 Status : KSYS_Status;
 prPress : REFTO REAL;
 pPressureLintab : REFTO KAPPL_LintabData;
 bNoPlaus : BOOL;
 pInjectOption : REFTO tOptionId;
 pPressureLintab2P : REFTO KAPPL_LintabData_2P;
 bHydraulic : BOOL;
 bExtPressControl : BOOL;
 bAIPressureLinked : BOOL;
END_VAR
#BEGIN_EDIT_BLOCK
// set lower limit 0.0 (no negative pressure allowed)
FPlausMaxInjectPressure.rLowerLimit := 0.0;

prPress := GET_SYNC_REFTO("Injection1.ai_Pressure", T#0s, Status);
bAIPressureLinked := (Status = KSYS_Status_OK);

//check if inject options (electric / hydraulic, external pressure control)
pInjectOption := GET_SYNC_REFTO('Injection1.sv_Options', T#0s, Status);
IF Status = KSYS_Status_OK THEN
   bHydraulic := (pInjectOption^ AND cOptionHydraulic) = cOptionHydraulic;
   bExtPressControl := (pInjectOption^ AND cSubOpExtPressControl) = cSubOpExtPressControl;
END_IF;

IF bAIPressureLinked OR bExtPressControl THEN
   IF bHydraulic THEN
      pPressureLintab2P := GET_SYNC_REFTO("Injection1.sv_PressureLintab", T#0s, Status);
      IF Status = KSYS_Status_OK THEN
         FPlausMaxInjectPressure.rUpperLimit := pPressureLintab2P^.LintabPoints.Point[2].rY;
      ELSE
         bNoPlaus := TRUE;
      END_IF;
   ELSE
      pPressureLintab := GET_SYNC_REFTO("Injection1.sv_PressureLintab", T#0s, Status);
      IF (Status = KSYS_Status_OK) AND (pPressureLintab^.LintabPoints.uNoOfPoints > 0) THEN
         FPlausMaxInjectPressure.rUpperLimit := pPressureLintab^.LintabPoints.Point[pPressureLintab^.LintabPoints.uNoOfPoints].rY;
      ELSE
         bNoPlaus := TRUE;
      END_IF;
   END_IF;
ELSE
   bNoPlaus := TRUE;
END_IF;

IF bNoPlaus THEN
   // set usefull limit, pressure higher 1000 bar problem with hydraulic hose, ...
   FPlausMaxInjectPressure.rUpperLimit := 999.0;
END_IF;

;#END_EDIT_BLOCK END_FUNCTION

#END_OF_IEC_PART

@Puma @IecEditor 6 131 @Pou 25
@@@BEG_Comment@@@

@@@END_Comment@@@

@BEG_Contents

@BEG_Func
@RT(17)FuncTreeContainer
2
@Var @RT(14)GET_SYNC_REFTO @RT(0) @T @T @DERIVED 0 @F @RT(22)KEBA_STANDARD_FUNCTION @F
@T
@BEG_Attrib
0 @RT(0) @RT(0)
@END_Attrib
1 1 @F @F @F @F

@Var @RT(9)IS_LINKED @RT(0) @T @T @DERIVED 0 @F @RT(22)KEBA_STANDARD_FUNCTION @F
@T
@BEG_Attrib
0 @RT(0) @RT(0)
@END_Attrib
1 1 @F @F @F @F

@END_Func

@BEG_Const
@RT(18)ConstTreeContainer
0
@END_Const

@BEG_Export

@BEG_Kind
@PLAUSIBILITY_FUNCTION @RT(23)FPlausMaxInjectPressure @STRUCTURED_TEXT
@RT(15)tsLimitDataReal @RT(0) @RT(0)
@END_Kind

@BEG_Dcl
@RT(16)DclTreeContainer
11
@Var @RT(11)DeviceClass @RT(0) @T @F @DT @RT(3)INT @RT(0) @T @T @BASIC 0 @F
@F @F
@T
@BEG_Attrib
3 @RT(0) @RT(0) @RT(0)
@END_Attrib
0 1 @F @F @F @F

@Var @RT(9)Userlevel @RT(0) @T @F @DT @RT(3)INT @RT(0) @T @T @BASIC 0 @F
@F @F
@T
@BEG_Attrib
3 @RT(0) @RT(0) @RT(0)
@END_Attrib
0 1 @F @F @F @F

@Var @RT(6)Status @RT(0) @T @T @DERIVED 0 @T @T @DT @RT(11)KSYS_Status @RT(0) @T @T @UNKNOWN 0 @F
@F @F
@T
@BEG_Attrib
3 @RT(0) @RT(0) @RT(0)
@END_Attrib
1 0 @F @F @F @F

@Var @RT(7)prPress @RT(0) @T @T @REFTO 0 @T @DT @RT(4)REAL @RT(0) @T @T @BASIC 0 @F
@F @F
@T
@BEG_Attrib
3 @RT(0) @RT(0) @RT(0)
@END_Attrib
1 0 @F @F @F @F

@Var @RT(15)pPressureLintab @RT(0) @T @T @REFTO 0 @F @DERIVED 0 @F @RT(16)KAPPL_LintabData @F
@T
@BEG_Attrib
3 @RT(0) @RT(0) @RT(0)
@END_Attrib
1 0 @F @F @F @F

@Var @RT(8)bNoPlaus @RT(0) @T @F @DT @RT(4)BOOL @RT(0) @T @T @BASIC 0 @F
@F @F
@T
@BEG_Attrib
3 @RT(0) @RT(0) @RT(0)
@END_Attrib
1 0 @F @F @F @F

@Var @RT(13)pInjectOption @RT(0) @T @T @REFTO 0 @F @DERIVED 0 @T @T @DT @RT(9)tOptionId @RT(0) @T @T @UNKNOWN 0 @F
@F @F
@T
@BEG_Attrib
3 @RT(0) @RT(0) @RT(0)
@END_Attrib
1 0 @F @F @F @F

@Var @RT(17)pPressureLintab2P @RT(0) @T @T @REFTO 0 @F @DERIVED 0 @F @RT(19)KAPPL_LintabData_2P @F
@T
@BEG_Attrib
3 @RT(0) @RT(0) @RT(0)
@END_Attrib
1 0 @F @F @F @F

@Var @RT(10)bHydraulic @RT(0) @T @F @DT @RT(4)BOOL @RT(0) @T @T @BASIC 0 @F
@F @F
@T
@BEG_Attrib
3 @RT(0) @RT(0) @RT(0)
@END_Attrib
1 0 @F @F @F @F

@Var @RT(16)bExtPressControl @RT(0) @T @F @DT @RT(4)BOOL @RT(0) @T @T @BASIC 0 @F
@F @F
@T
@BEG_Attrib
3 @RT(0) @RT(0) @RT(0)
@END_Attrib
1 0 @F @F @F @F

@Var @RT(17)bAIPressureLinked @RT(0) @T @F @DT @RT(4)BOOL @RT(0) @T @T @BASIC 0 @F
@F @F
@T
@BEG_Attrib
3 @RT(0) @RT(0) @RT(0)
@END_Attrib
1 0 @F @F @F @F

@END_Dcl

@END_Export

@BEG_Body
@TL(38)
// set lower limit 0.0 (no negative pressure allowed)
FPlausMaxInjectPressure.rLowerLimit := 0.0;

prPress := GET_SYNC_REFTO("Injection1.ai_Pressure", T#0s, Status);
bAIPressureLinked := (Status = KSYS_Status_OK);

//check if inject options (electric / hydraulic, external pressure control)
pInjectOption := GET_SYNC_REFTO('Injection1.sv_Options', T#0s, Status);
IF Status = KSYS_Status_OK THEN
   bHydraulic := (pInjectOption^ AND cOptionHydraulic) = cOptionHydraulic;
   bExtPressControl := (pInjectOption^ AND cSubOpExtPressControl) = cSubOpExtPressControl;
END_IF;

IF bAIPressureLinked OR bExtPressControl THEN
   IF bHydraulic THEN
      pPressureLintab2P := GET_SYNC_REFTO("Injection1.sv_PressureLintab", T#0s, Status);
      IF Status = KSYS_Status_OK THEN
         FPlausMaxInjectPressure.rUpperLimit := pPressureLintab2P^.LintabPoints.Point[2].rY;
      ELSE
         bNoPlaus := TRUE;
      END_IF;
   ELSE
      pPressureLintab := GET_SYNC_REFTO("Injection1.sv_PressureLintab", T#0s, Status);
      IF (Status = KSYS_Status_OK) AND (pPressureLintab^.LintabPoints.uNoOfPoints > 0) THEN
         FPlausMaxInjectPressure.rUpperLimit := pPressureLintab^.LintabPoints.Point[pPressureLintab^.LintabPoints.uNoOfPoints].rY;
      ELSE
         bNoPlaus := TRUE;
      END_IF;
   END_IF;
ELSE
   bNoPlaus := TRUE;
END_IF;

IF bNoPlaus THEN
   // set usefull limit, pressure higher 1000 bar problem with hydraulic hose, ...
   FPlausMaxInjectPressure.rUpperLimit := 999.0;
END_IF;

@END_Body

@END_Contents

(* ---- FPlausMaxSysPressure.pu ---- *)
IMPORT_OVER_LISTFILE
 GET_SYNC_REFTO
, IS_LINKED
, tsLimitDataReal
, KSYS_Status
, KAPPL_LintabData_2P

END_IMPORT

PLAUSIBILITY_FUNCTION FPlausMaxSysPressure : tsLimitDataReal

VAR_INPUT
 DeviceClass : INT;
 Userlevel : INT;
END_VAR

VAR
 Status : KSYS_Status;
 prSysPress : REFTO REAL;
 pSysPressureLintab : REFTO KAPPL_LintabData_2P;
 bNoPlaus : BOOL;
END_VAR
#BEGIN_EDIT_BLOCK
// set lower limit 0.0 (no negative pressure allowed)
FPlausMaxSysPressure.rLowerLimit := 0.0;

prSysPress := GET_SYNC_REFTO("Injection1.ai_SysPressure", T#0s, Status);
IF Status = KSYS_Status_OK THEN
   pSysPressureLintab := GET_SYNC_REFTO("Injection1.sv_SysPressureLintab", T#0s, Status);
   IF Status = KSYS_Status_OK THEN
      IF pSysPressureLintab^.LintabPoints.uNoOfPoints > 0 THEN
         FPlausMaxSysPressure.rUpperLimit := pSysPressureLintab^.LintabPoints.Point[pSysPressureLintab^.LintabPoints.uNoOfPoints].rY;
      ELSE
         bNoPlaus := TRUE;
      END_IF;
   ELSE
      bNoPlaus := TRUE;
   END_IF;
ELSE
   bNoPlaus := TRUE;
END_IF;
IF bNoPlaus THEN
   // set usefull limit, pressure higher 1000 bar problem with hydraulic hose, ...
   FPlausMaxSysPressure.rUpperLimit := 999.0;
END_IF;

;#END_EDIT_BLOCK END_FUNCTION

#END_OF_IEC_PART

@Puma @IecEditor 6 131 @Pou 25
@@@BEG_Comment@@@

@@@END_Comment@@@

@BEG_Contents

@BEG_Func
@RT(17)FuncTreeContainer
2
@Var @RT(14)GET_SYNC_REFTO @RT(0) @T @T @DERIVED 0 @F @RT(22)KEBA_STANDARD_FUNCTION @F
@T
@BEG_Attrib
0 @RT(0) @RT(0)
@END_Attrib
1 1 @F @F @F @F

@Var @RT(9)IS_LINKED @RT(0) @T @T @DERIVED 0 @F @RT(22)KEBA_STANDARD_FUNCTION @F
@T
@BEG_Attrib
0 @RT(0) @RT(0)
@END_Attrib
1 1 @F @F @F @F

@END_Func

@BEG_Const
@RT(18)ConstTreeContainer
0
@END_Const

@BEG_Export

@BEG_Kind
@PLAUSIBILITY_FUNCTION @RT(20)FPlausMaxSysPressure @STRUCTURED_TEXT
@RT(15)tsLimitDataReal @RT(0) @RT(0)
@END_Kind

@BEG_Dcl
@RT(16)DclTreeContainer
6
@Var @RT(11)DeviceClass @RT(0) @T @F @DT @RT(3)INT @RT(0) @T @T @BASIC 0 @F
@F @F
@T
@BEG_Attrib
3 @RT(0) @RT(0) @RT(0)
@END_Attrib
0 1 @F @F @F @F

@Var @RT(9)Userlevel @RT(0) @T @F @DT @RT(3)INT @RT(0) @T @T @BASIC 0 @F
@F @F
@T
@BEG_Attrib
3 @RT(0) @RT(0) @RT(0)
@END_Attrib
0 1 @F @F @F @F

@Var @RT(6)Status @RT(0) @T @T @DERIVED 0 @T @T @DT @RT(11)KSYS_Status @RT(0) @T @T @UNKNOWN 0 @F
@F @F
@T
@BEG_Attrib
3 @RT(0) @RT(0) @RT(0)
@END_Attrib
1 0 @F @F @F @F

@Var @RT(10)prSysPress @RT(0) @T @T @REFTO 0 @T @DT @RT(4)REAL @RT(0) @T @T @BASIC 0 @F
@F @F
@T
@BEG_Attrib
3 @RT(0) @RT(0) @RT(0)
@END_Attrib
1 0 @F @F @F @F

@Var @RT(18)pSysPressureLintab @RT(0) @T @T @REFTO 0 @F @DERIVED 0 @F @RT(19)KAPPL_LintabData_2P @F
@T
@BEG_Attrib
3 @RT(0) @RT(0) @RT(0)
@END_Attrib
1 0 @F @F @F @F

@Var @RT(8)bNoPlaus @RT(0) @T @F @DT @RT(4)BOOL @RT(0) @T @T @BASIC 0 @F
@F @F
@T
@BEG_Attrib
3 @RT(0) @RT(0) @RT(0)
@END_Attrib
1 0 @F @F @F @F

@END_Dcl

@END_Export

@BEG_Body
@TL(24)
// set lower limit 0.0 (no negative pressure allowed)
FPlausMaxSysPressure.rLowerLimit := 0.0;

prSysPress := GET_SYNC_REFTO("Injection1.ai_SysPressure", T#0s, Status);
IF Status = KSYS_Status_OK THEN
   pSysPressureLintab := GET_SYNC_REFTO("Injection1.sv_SysPressureLintab", T#0s, Status);
   IF Status = KSYS_Status_OK THEN
      IF pSysPressureLintab^.LintabPoints.uNoOfPoints > 0 THEN
         FPlausMaxSysPressure.rUpperLimit := pSysPressureLintab^.LintabPoints.Point[pSysPressureLintab^.LintabPoints.uNoOfPoints].rY;
      ELSE
         bNoPlaus := TRUE;
      END_IF;
   ELSE
      bNoPlaus := TRUE;
   END_IF;
ELSE
   bNoPlaus := TRUE;
END_IF;
IF bNoPlaus THEN
   // set usefull limit, pressure higher 1000 bar problem with hydraulic hose, ...
   FPlausMaxSysPressure.rUpperLimit := 999.0;
END_IF;

@END_Body

@END_Contents
